(* IEC 61131-3 sources: LASAL/Class/XXXBase_IOs, 1 file *)

(* ---- XXXBase_IOs.st ---- *)
(*!
<Class
	Name               = "XXXBase_IOs"
	Revision           = "1.0"
	RealtimeTask       = "false"
	CyclicTask         = "false"
	BackgroundTask     = "false"
	Sigmatek           = "true"
	OSInterface        = "false"
	HighPriority       = "false"
	Automatic          = "false"
	UpdateMode         = "Prescan"
	IconPath           = ".\Class\DigInOut.ICO"
	SharedCommandTable = "true"
	Objectsize         = "(570,540)"
	Comment            = "Baseclass for CPU_IO classes.">
	<Channels>
		<Server Name="CAN_1_Connect" Class="_CanLib" Visualized="false" Initialize="false" WriteProtected="true" Retentive="false" Comment="Connection servers for Hardware-Editor."/>
		<Server Name="CAN_2_Connect" Class="_CanLib" Visualized="false" Initialize="false" WriteProtected="true" Retentive="false" Comment="Connection servers for Hardware-Editor."/>
		<Server Name="ClassState" Visualized="true" Initialize="false" WriteProtected="true" Retentive="false" Comment="Shows the state of the class.&#13;&#10;0 ... ok."/>
		<Server Name="COM_1_Connect" Class="_SerLib" Visualized="false" Initialize="false" WriteProtected="true" Retentive="false" Comment="Connection servers for Hardware-Editor."/>
		<Server Name="COM_2_Connect" Class="_SerLib" Visualized="false" Initialize="false" WriteProtected="true" Retentive="false" Comment="Connection servers for Hardware-Editor."/>
		<Server Name="USB_1_Connect" Visualized="false" Initialize="false" WriteProtected="true" Retentive="false" Comment="Connection servers for Hardware-Editor."/>
		<Client Name="_CanLib1" Required="true" Internal="true"/>
		<Client Name="_CanLib2" Required="true" Internal="true"/>
		<Client Name="_SerLib1" Required="true" Internal="true"/>
		<Client Name="_SerLib2" Required="true" Internal="true"/>
		<Client Name="To_HwControl" Required="true" Internal="false" Comment="Connect to Client &quot;Control&quot; of &quot;HwControl&quot;-Object"/>
	</Channels>
	<RevDoku>
		<Owner Company="Sigmatek" Author="HaeTho"/>
		<Dokumentation Revision="1.0" Date="02.08.2018" Author="HaeTho" Company="Sigmatek" Description="Hardware-Editor Bus-Connectors, first library version"/>
	</RevDoku>
	<Network Name="XXXBase_IOs">
		<!-- List of Components in this network -->
		<Components>
			<Object
				Name       = "_CanLib1"
				Class      = "_CanLib"
				Position   = "(150,300)"
				Visualized = "true"
				Remotely   = "true">
				<Channels>
					<Server Name="CanBus" Value="0"/>
					<Server Name="Command"/>
					<Client Name="To_Can"/>
				</Channels>
			</Object>
			<Object
				Name       = "_CanLib2"
				Class      = "_CanLib"
				Position   = "(150,510)"
				Visualized = "true"
				Remotely   = "true">
				<Channels>
					<Server Name="CanBus" Value="1"/>
					<Server Name="Command"/>
					<Client Name="To_Can"/>
				</Channels>
			</Object>
			<Object
				Name       = "_SerLib1"
				Class      = "_SerLib"
				Position   = "(150,720)"
				Visualized = "true"
				Remotely   = "true">
				<Channels>
					<Server Name="Com" Value="0"/>
					<Server Name="Command"/>
				</Channels>
			</Object>
			<Object
				Name       = "_SerLib2"
				Class      = "_SerLib"
				Position   = "(150,930)"
				Visualized = "true"
				Remotely   = "true">
				<Channels>
					<Server Name="Com" Value="1"/>
					<Server Name="Command"/>
				</Channels>
			</Object>
		</Components>
		<Comments>
		</Comments>
		<!-- List of Connections in this network -->
		<Connections>
			<Connection Source="this._CanLib1" Destination="_CanLib1.Command"/>
			<Connection Source="this.CAN_1_Connect" Destination="_CanLib1.Command" Vertices="(652,330),(480,390),"/>
			<Connection Source="this._CanLib2" Destination="_CanLib2.Command"/>
			<Connection Source="this.CAN_2_Connect" Destination="_CanLib2.Command" Vertices="(652,390),(480,600),"/>
			<Connection Source="this._SerLib1" Destination="_SerLib1.Command"/>
			<Connection Source="this.COM_1_Connect" Destination="_SerLib1.Command" Vertices="(652,450),(450,810),"/>
			<Connection Source="this._SerLib2" Destination="_SerLib2.Command"/>
			<Connection Source="this.COM_2_Connect" Destination="_SerLib2.Command" Vertices="(652,510),(450,1020),"/>
		</Connections>
		<!-- Headerfiles -->
		<Options>
		</Options>
	</Network>
</Class>
*)
XXXBase_IOs : CLASS
  //Servers:
	ClassState 	: SvrChCmd_DINT;
	USB_1_Connect 	: SvrChCmd_DINT;
	CAN_1_Connect 	: SvrChCmd_DINT;
	CAN_2_Connect 	: SvrChCmd_DINT;
	COM_1_Connect 	: SvrChCmd_DINT;
	COM_2_Connect 	: SvrChCmd_DINT;
  //Clients:
	To_HwControl 	: CltChCmd_HwControl;
	_SerLib1 	: CltChCmd__SerLib;
	_SerLib2 	: CltChCmd__SerLib;
	_CanLib1 	: CltChCmd__CanLib;
	_CanLib2 	: CltChCmd__CanLib;
  //Variables:
  //Functions:
  //Tables:
	FUNCTION @STD
		VAR_OUTPUT
			ret_code	: CONFSTATES;
		END_VAR;
	FUNCTION GLOBAL TAB @CT_;
END_CLASS;

#pragma using _CanLib
#pragma using _SerLib
#pragma usingLtd HwControl
